PROGRAM MAIN
VAR
	bLed1 AT %Q*: BOOL := FALSE;
	
	BButton1 AT %I*: BOOL := false;
	bButton2 AT %I*: BOOL := FALSE;
	bButton3 AT %I*: BOOL := FALSE;
	
	bTriggerLong: BOOL;
	bTriggerShort: BOOL;
	
	FB_Timer_Setting: CTUD ;
	fbtimer: TON;
	FB_Button: FB_ShortLongClick;
	FB_Lights: FB_Light;
	fbWarning: TOF;
	fbBlinking: TOF;
	fbTON: TON := (PT := TIME#100MS);
	bLED2 AT %Q*: BOOL;
END_VAR

FB_Button(bSwitch:= BButton1, tSwitchTime:= T#2S, bShortClick=> bTriggerShort , bLongClick=> bTriggerLong);
FB_Lights(bOn:=  , bOff:= fbtimer.q, bToggle:= bTriggerShort, bLight=>bLed1 );
FB_Timer_Setting(CU:= bButton2, CD:= bButton3 );
fbtimer(IN:= bLed1 AND NOT bTriggerLong , PT:=  TO_TIME(FB_Timer_Setting.CV * 1000 + 3*1000));
fbWarning(IN:= bTriggerShort OR bTriggerLong , PT:= TO_TIME(FB_Timer_Setting.CV * 1000));
fbBlinking(IN:= fbWarning.Q, PT:= T#3S);
IF (NOT fbWarning.Q AND bLed1) AND fbBlinking.Q THEN
	fbTON(IN:= NOT(fbTON.Q), Q=>bLED2);
END_IF

END_PROGRAM

(* stored: Version 1.1.0.1, ProductVersion 3.1.4024.12
   POU MAIN: Id {9089100c-cffe-410f-b8bd-6937b0c975f5}, SpecialFunc None *)
